(*

## Short summary

This class provides assert statements the most common data:
It implements the interface `IAssertions`
For ``STRUCT``, ``ARRAY``, ``FUNCTION BLOCK``, ``ENUM``  use `Assertions.binary`
For ``BYTE``, ``WORD``, ``DWORD``, ``LWORD``, ``__XWORD`` use `Assertions.bitNumber`
For ``BOOL`` use `Assertions.boolean`
For ``DT``, ``TOD``, ``DATE`` use `Assertions.dateAndTime`
For ``REAL``, ``LREAL`` use `Assertions.float`
For ``SINT``, ``INT``, ``DINT``, ``LINT``, ``__XINT`` use `Assertions.integer`
For ``CNM_AbsrtractObject.IObject`` use `Assertions.object`
For ``POINTER`` use `Assertions.pointers`
For ``STRING``, ``WSTRING`` use `Assertions.strings`
For ``TIME``, ``LTIME`` use `Assertions.times`

.. <legal notes>

legal notes
=================
| SPDX-FileCopyrightText: © 2022 ekvip automation GmbH <info@ekvip.de>
| SPDX-License-Identifier: Apache-2.0
| For details check: Apache-2.0_

.. _Apache-2.0: https://www.apache.org/licenses/LICENSE-2.0

.. </legal notes>



*)

{attribute 'reflection'}
FUNCTION_BLOCK INTERNAL Assertions EXTENDS CNM_AbstractObject.Object IMPLEMENTS IAssertions, IAssertCallBacksetter
VAR
	(* class to handle binary assertions *)
	binaryAssertions	:BinaryAssertions();
	(* class to handle bit number assertions *)
	bitNumberAssertions	:BitNumberAssertions();
	(* class to handle boolean assertions *)
	booleanAssertions	:BooleanAssertion();
	(* class to handle date and time assertions *)
	dateTimeAssertions	:DateAndTimeAssertions();
	(* class to handle float assertions *)
	floatAssertions		:FloatAssertions();
	(* class to handle integer assertions *)
	integerAssertions	:IntegerAssertions();
	(* class to handle object assertions *)
	objectAssertions	:ObjectAssertions();
	(* class to handle pointer assertions *)
	pointerAssertions	:PointerAssertions();
	(* class to handle string assertions *)
	stringAssertions	:StringAssertions();
	(* class to handle time assertions *)
	timeAssertions		:TimeAssertions();
END_VAR

(*

## Short summary
Returns the interface `IBinaryAssertions`
with assert statements for binary data 

.. <legal notes>

legal notes
=================
| SPDX-FileCopyrightText: © 2022 ekvip automation GmbH <info@ekvip.de>
| SPDX-License-Identifier: Apache-2.0
| For details check: Apache-2.0_

.. _Apache-2.0: https://www.apache.org/licenses/LICENSE-2.0

.. </legal notes>

*)

PROPERTY binary :IBinaryAssertions
GET
binary := THIS^.binaryAssertions;
END_GET
END_PROPERTY

(*

## Short summary
Returns the interface `IBitNumberAssertions`
with assert statements for bit numbers 

.. <legal notes>

legal notes
=================
| SPDX-FileCopyrightText: © 2022 ekvip automation GmbH <info@ekvip.de>
| SPDX-License-Identifier: Apache-2.0
| For details check: Apache-2.0_

.. _Apache-2.0: https://www.apache.org/licenses/LICENSE-2.0

.. </legal notes>

*)

PROPERTY bitNumber :IBitNumberAssertions
GET
bitNumber := THIS^.bitNumberAssertions;
END_GET
END_PROPERTY

(*

## Short summary
Returns the interface `IBooleanAssertion`
with assert statements for booleans

.. <legal notes>

legal notes
=================
| SPDX-FileCopyrightText: © 2022 ekvip automation GmbH <info@ekvip.de>
| SPDX-License-Identifier: Apache-2.0
| For details check: Apache-2.0_

.. _Apache-2.0: https://www.apache.org/licenses/LICENSE-2.0

.. </legal notes>

*)

PROPERTY boolean :IBooleanAssertion
GET
boolean := THIS^.booleanAssertions;
END_GET
END_PROPERTY

(*

## Short summary
This abstract property returns the class name of the concrete object, 
It's for debugging purpose

.. <legal notes>

legal notes
=================
| SPDX-FileCopyrightText: © 2022 ekvip automation GmbH <info@ekvip.de>
| SPDX-License-Identifier: Apache-2.0
| For details check: Apache-2.0_

.. _Apache-2.0: https://www.apache.org/licenses/LICENSE-2.0

.. </legal notes>

*)

PROPERTY className :CNM_AbstractObject.ClassName
GET
className := 'CNM_Assertor.Assertions';
END_GET
END_PROPERTY

(*

## Short summary
Returns the interface `IDateAndTimeAssertions`
with assert statements for date and time data types

.. <legal notes>

legal notes
=================
| SPDX-FileCopyrightText: © 2022 ekvip automation GmbH <info@ekvip.de>
| SPDX-License-Identifier: Apache-2.0
| For details check: Apache-2.0_

.. _Apache-2.0: https://www.apache.org/licenses/LICENSE-2.0

.. </legal notes>

*)

PROPERTY dateAndTime :IDateAndTimeAssertions
GET
dateAndTime := THIS^.dateTimeAssertions;
END_GET
END_PROPERTY

(*

## Short summary
Returns the interface `IFloatAssertions`
with assert statements for floatings

.. <legal notes>

legal notes
=================
| SPDX-FileCopyrightText: © 2022 ekvip automation GmbH <info@ekvip.de>
| SPDX-License-Identifier: Apache-2.0
| For details check: Apache-2.0_

.. _Apache-2.0: https://www.apache.org/licenses/LICENSE-2.0

.. </legal notes>

*)

PROPERTY float :IFloatAssertions
GET
float := THIS^.floatAssertions;
END_GET
END_PROPERTY

(*

## Short summary
Returns the interface `IIntergerAssertions`
with assert statements for integers

.. <legal notes>

legal notes
=================
| SPDX-FileCopyrightText: © 2022 ekvip automation GmbH <info@ekvip.de>
| SPDX-License-Identifier: Apache-2.0
| For details check: Apache-2.0_

.. _Apache-2.0: https://www.apache.org/licenses/LICENSE-2.0

.. </legal notes>

*)

PROPERTY integer :IIntegerAssertions
GET
integer := THIS^.integerAssertions;
END_GET
END_PROPERTY

(*

## Short summary
Returns the interface `IObjectAssertions`
with assert statements for ``CNM_AbstractObject.IObject``

.. <legal notes>

legal notes
=================
| SPDX-FileCopyrightText: © 2022 ekvip automation GmbH <info@ekvip.de>
| SPDX-License-Identifier: Apache-2.0
| For details check: Apache-2.0_

.. _Apache-2.0: https://www.apache.org/licenses/LICENSE-2.0

.. </legal notes>

*)

PROPERTY object :IObjectAssertions
GET
object := THIS^.objectAssertions;
END_GET
END_PROPERTY

(*

## Short summary
Returns the interface `IPointerAssertions`
with assert statements for pointers

.. <legal notes>

legal notes
=================
| SPDX-FileCopyrightText: © 2022 ekvip automation GmbH <info@ekvip.de>
| SPDX-License-Identifier: Apache-2.0
| For details check: Apache-2.0_

.. _Apache-2.0: https://www.apache.org/licenses/LICENSE-2.0

.. </legal notes>

*)

PROPERTY pointers :IPointerAssertions
GET
pointers := THIS^.pointerAssertions;
END_GET
END_PROPERTY

(*

## Short summary
This methods is the setter for the callback class if an assertion was false

.. <legal notes>

legal notes
=================
| SPDX-FileCopyrightText: © 2022 ekvip automation GmbH <info@ekvip.de>
| SPDX-License-Identifier: Apache-2.0
| For details check: Apache-2.0_

.. _Apache-2.0: https://www.apache.org/licenses/LICENSE-2.0

.. </legal notes>



*)

METHOD setCallBack
VAR_INPUT
	(* the class that must be informed if an assertion is false *)
	callBack	:IAssertCallBack;  
END_VAR
THIS^.binaryAssertions.setCallBack(callBack);
THIS^.bitNumberAssertions.setCallBack(callBack);
THIS^.booleanAssertions.setCallBack(callBack);
THIS^.dateTimeAssertions.setCallBack(callBack);
THIS^.floatAssertions.setCallBack(callBack);
THIS^.integerAssertions.setCallBack(callBack);
THIS^.objectAssertions.setCallBack(callBack);
THIS^.pointerAssertions.setCallBack(callBack);
THIS^.stringAssertions.setCallBack(callBack);
THIS^.timeAssertions.setCallBack(callBack);
END_METHOD

(*

## Short summary
Returns the interface `IStringAssertions`
with assert statements for windows-1252 and UTF-16 strings

.. <legal notes>

legal notes
=================
| SPDX-FileCopyrightText: © 2022 ekvip automation GmbH <info@ekvip.de>
| SPDX-License-Identifier: Apache-2.0
| For details check: Apache-2.0_

.. _Apache-2.0: https://www.apache.org/licenses/LICENSE-2.0

.. </legal notes>

*)

PROPERTY strings :IStringAssertions
GET
strings := THIS^.stringAssertions;
END_GET
END_PROPERTY

(*

## Short summary
Returns the interface `ITimeAssertions`
with assert statements for time data types

.. <legal notes>

legal notes
=================
| SPDX-FileCopyrightText: © 2022 ekvip automation GmbH <info@ekvip.de>
| SPDX-License-Identifier: Apache-2.0
| For details check: Apache-2.0_

.. _Apache-2.0: https://www.apache.org/licenses/LICENSE-2.0

.. </legal notes>

*)

PROPERTY times :ITimeAssertions
GET
times := THIS^.timeAssertions;
END_GET
END_PROPERTY

END_FUNCTION_BLOCK

(* stored: Version 1.1.0.1, ProductVersion 3.1.4026.12
   POU Assertions: Id {6a4a64d5-6ec4-4b4b-aade-c47eac3c5641}, SpecialFunc None
   Property binary: Id {142c926b-7501-4ccc-8f69-6a247de43135}
   Get Get: Id {b7c2278f-bedb-4fab-91a7-77f4c4281a99}
   Property bitNumber: Id {4ec29991-655d-4950-a714-b3d8ba0255ee}
   Get Get: Id {2f73ad81-d28d-45ba-8ce6-a07d77138d29}
   Property boolean: Id {acd9bbbe-07df-4677-bb51-c2cdfa44c9d6}
   Get Get: Id {945c8e76-685f-488e-94b6-80134f6cfdc8}
   Property className: Id {86f6a553-7cca-4892-be2a-c6d1aced52d5}
   Get Get: Id {1662ac8b-568f-45a9-95f2-17365adef5d5}
   Property dateAndTime: Id {55de2bbc-cb36-431d-9a9e-da75b292109b}
   Get Get: Id {a9147822-4b63-4e17-ac59-4495fa4e47de}
   Property float: Id {9218355c-182a-4f47-b7f0-8992a0809776}
   Get Get: Id {4c4a36ad-c249-406f-aa81-bd04408b6b84}
   Property integer: Id {b65a6d6b-b495-4f3b-95a2-c7861bb5407d}
   Get Get: Id {cbc086f1-96e9-43ab-ab5f-e9f32d1cea0c}
   Property object: Id {7bf60662-43d8-4e19-adbd-cccbf5d058bf}
   Get Get: Id {9c5cd401-d750-43b6-af55-add2be37063f}
   Property pointers: Id {6724e1cf-e6cb-4515-9765-00eb60337b3b}
   Get Get: Id {5be8d647-99ca-4d89-9fbf-1876130341c5}
   Method setCallBack: Id {3f4eb8e9-9028-4ea0-b455-29d500d57685}
   Property strings: Id {63ab39da-e661-4a29-8ea2-a177aebf05fb}
   Get Get: Id {98e545e1-86cb-4f6a-a67c-fa23903f6378}
   Property times: Id {07e8307b-c360-425a-acd8-547c6726db30}
   Get Get: Id {b856cf7a-028c-4686-b2f9-e0dcd58f45fe} *)
